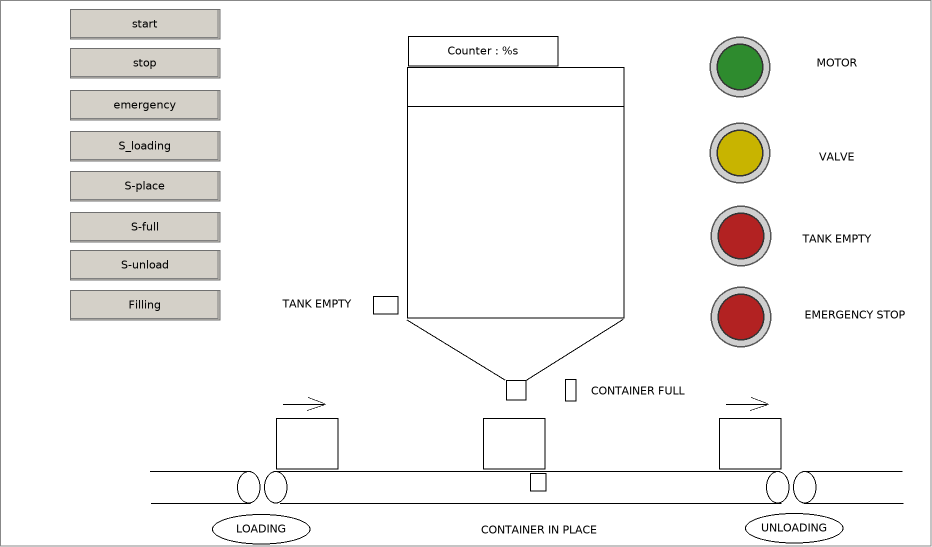
VISUALIZATION Visualization  // 932x547
    Lamp1 (705,32 70x70), variable: LADDER1.Motor, style: Lamp-Lamp1-Green
    Button (70,9 150x30), "start"
        OnMouseDown: toggle LADDER1.start
    Button (70,48 150x30), "stop"
        OnMouseDown: toggle LADDER1.stop
    Button (70,212 150x30), "S-full"
        OnMouseDown: toggle LADDER1.S_full
    Button (70,171 150x30), "S-place"
        OnMouseDown: toggle LADDER1.S_place
    Button (70,90 150x30), "emergency"
        OnMouseDown: toggle LADDER1.emergency
    Lamp1 (705,118 70x70), variable: LADDER1.valve, style: Lamp-Lamp1-Yellow
    Lamp1 (706,201 70x70), variable: LADDER1.TankEmpty, style: Lamp-Lamp1-Red
    Button (70,250 150x30), "S-unload"
        OnMouseDown: toggle LADDER1.S_unload
    Button (70,131 150x30), "S_loading"
        OnMouseDown: toggle LADDER1.S_loading
    Button (70,290 150x30), "Filling"
        OnMouseDown: toggle LADDER1.FILLING
    Rectangle (407,67 217x251)
    Rectangle (407,106 217x212), invisible if: LADDER1.TankEmpty
    Line (413,321)
    Line (505,380) (407,320)
    Line (585,354)
    Line (526,380) (623,319)
    Rectangle (506,380 20x20)
    Rectangle (483,418 62x51), colour toggle: LADDER1.S_full
        OnMouseDown: toggle LADDER1.S_full
    Rectangle (276,418 62x51)
    Rectangle (719,418 62x51)
    Line (726,404) (767,404)
    Line (751,397) (767,403)
    Line (750,410) (768,404)
    Line (283,404) (324,404)
    Line (308,397) (324,403)
    Line (307,410) (325,404)
    Ellipse (264,471 23x32)
    Line (278,471) (779,471)
    Ellipse (766,471 23x32)
    Line (280,503) (781,503)
    Ellipse (237,471 23x32)
    Ellipse (793,471 23x32)
    Line (803,471) (902,471)
    Line (804,503) (903,503)
    Line (150,471) (249,471)
    Line (151,503) (250,503)
    Ellipse (212,514 98x30), "LOADING"
    Ellipse (745,513 98x30), "UNLOADING"
    Rectangle (530,473 16x18)
    Rectangle (565,379 11x22)
    Label (549,376 178x30), "CONTAINER FULL"
    Label (464,515 150x30), "CONTAINER IN PLACE"
    Label (750,42 174x42), "MOTOR"
    Label (750,136 174x42), "VALVE"
    Label (750,218 174x42), "TANK EMPTY"
    Label (242,289 150x30), "TANK EMPTY"
    Rectangle (373,296 25x18)
    Rectangle (408,36 150x30), "Counter : %s", text variable: MAIN.LADDER1.counter.CV
    Lamp1 (706,282 70x70), variable: LADDER1.emergency, style: Lamp-Lamp1-Red
    Label (780,300 150x30), "EMERGENCY STOP"
END_VISUALIZATION

(* stored: Version 1.1.0.1, ProductVersion 3.1.4020.12
   Visu Visualization: Id {89b6d401-b465-4148-8687-009c3905fc00} *)
